// TIA Portal V19 export
DATA_BLOCK "A0304_Manager"   // DB99
// stored: InstanceOfName A0304_Manager_FB, InstanceOfType FB
"A0304_Manager_FB"
   // VAR_INPUT
   //    AreaInterface : "AreaInterface";
   //    ZSI : "udt_ZoneSafetyInterface";
   //    DataIn : Struct
   //       PbScaricaPacco : Bool;
   //       PbReggiaturaConclusa : Bool;
   //       LsMatPres1Load : Bool;
   //       LsMatPres2Load : Bool;
   //       LsMatPres1UnLoad : Bool;
   //       LsMatPres2UnLoad : Bool;
   //    END_STRUCT;
   //    CIn : Struct
   //       Navetta : Struct
   //          Testa : Struct
   //             Ax : "Positioning_DOL_Machine_COut";
   //             PalettiEsterni : "ValveMachine_COut";
   //             PalettiInterni : "ValveMachine_COut";
   //          END_STRUCT;
   //          Coda : Struct
   //             Ax : "Positioning_DOL_Machine_COut";
   //             PalettiEsterni : "ValveMachine_COut";
   //             PalettiInterni : "ValveMachine_COut";
   //          END_STRUCT;
   //          Cumulativo : Struct
   //             PalettiEsterni : "ValveMachine_COut";
   //             PalettiInterni : "ValveMachine_COut";
   //          END_STRUCT;
   //          ReadyToRecive : Bool;
   //       END_STRUCT;
   //       Sollevamento : Struct
   //          ReadyToDrop : Bool;
   //       END_STRUCT;
   //       Antiribaltamento : Struct
   //          Work : Bool;
   //          Rest : Bool;
   //          PalettoPos0 : Bool;
   //       END_STRUCT;
   //       Manager03 : Struct
   //          IsWaiting_NoPiecesBefore : Bool;
   //       END_STRUCT;
   //       ProdManager : "Prod_Beam_Ctrl";
   //    END_STRUCT;
   // END_VAR
   // VAR_OUTPUT
   //    COut { ExternalAccessible := 'False'; ExternalVisible := 'False'; ExternalWritable := 'False'} : Struct
   //       Navetta : Struct
   //          EnableStopDoorOpeningReq : Bool;
   //          EnableStopInPhase : Bool;
   //          EnableStopProgrammed : Bool;
   //          Control_ON : Bool;
   //          CanMoveFreely : Bool;
   //          OP : Struct
   //             VAI_A_PRELIEVO : Bool;
   //             PRELIEVO : Bool;
   //             VAI_A_DEPOSITO : Bool;
   //             DEPOSITO : Bool;
   //          END_STRUCT;
   //       END_STRUCT;
   //       Sollevatore : Struct
   //          ReadyToRecive : Bool;
   //          OutOfWorkspace : Bool;
   //       END_STRUCT;
   //    END_STRUCT;
   //    MachineInterface : "MachineInterface";
   // END_VAR
   // VAR_IN_OUT
   //    Par_Navetta : Struct
   //       PosPrePrelievo : LReal;
   //       PosPrelievo : LReal;
   //       PosDeposito : LReal;
   //       ToleranceWindow : LReal;
   //    END_STRUCT;
   // END_VAR
   // VAR
   //    Alarm : Struct
   //       ShuttleNotEmpty : Bool;
   //       STOP_FineTurno : Bool;
   //       STOP_ControlloQualita : Bool;
   //       STOP_End_Of_Proroduction : Bool;
   //       TimeoutRimozionePaccoMES : Bool;
   //    END_STRUCT;
   //    Warning : Struct
   //       UnloadNotPossible : Bool;
   //       TimeoutRimozionePaccoMES : Bool;
   //    END_STRUCT;
   //    OP_CND : Struct
   //       VaiAPrelievo : Array[0..15] of "OpCnd";
   //       Prelievo { S7_SetPoint := 'True'} : Array[0..15] of "OpCnd";
   //       VaiADeposito : Array[0..15] of "OpCnd";
   //       Deposito : Array[0..15] of "OpCnd";
   //    END_STRUCT;
   //    Sts : Struct
   //       SemiAut : Struct
   //          ON : Bool;
   //          PbMaterialFwd : Bool;
   //          Request : Bool;
   //       END_STRUCT;
   //       InPosDeposito : Bool;
   //       InPosPrePrelievo : Bool;
   //       InPosPrelievo : Bool;
   //       RichiestaVaiDeposito : Bool;
   //       RichiestaVaiPrelievo : Bool;
   //       IsStandstill : Bool;
   //       AlarmsPresence : Bool;
   //       WarningsPresence : Bool;
   //    END_STRUCT;
   //    Ctrl : Struct
   //       Cycle : Struct
   //          VaiAPrelievo : Bool;
   //          Prelievo : Bool;
   //          VaiADeposito : Bool;
   //          Deposito : Bool;
   //       END_STRUCT;
   //       ReggiaturaConclusa : Bool;
   //       ConfermaPaccoScaricato : Bool;
   //       Stop : Bool;
   //    END_STRUCT;
   //    AUX : Struct
   //       SemiAut_Pb : Bool;
   //       PbScaricaPacco : Bool;
   //       PbReggiaturaConclusa : Bool;
   //    END_STRUCT;
   //    TON_MatPres : IEC_TIMER;
   //    TON_Stop : IEC_TIMER;
   //    TON_ForceConfermaPaccoScraicato : IEC_TIMER;
   //    TON_TimeoutRimozionePaccoMES { S7_SetPoint := 'True'} : IEC_TIMER;
   //    TON_WngTimeoutRimozionePaccoMES { S7_SetPoint := 'True'} : IEC_TIMER;
   //    CycleWithShortPiece : Bool;
   // END_VAR
BEGIN
END_DATA_BLOCK
